// TIA Portal V20 export
FUNCTION_BLOCK "Sequence_1_TopTapeLoading"   // FB32851, LAD
TITLE = Sequence
// Sequence template programmend in ladder logic
// stored: IsIECCheckEnabled true, MemoryReserve 100, Namespace Unit1.Em3, SetENOAutomatically true
   VAR_INPUT
      unitStatus : "LAF_typeUnitStatus";
   END_VAR
   VAR
      instSequenceLADControl { ExternalWritable := 'False'} : "LAF_ControlLadSequence";
      instSequenceLADStatus { ExternalWritable := 'False'} : "LAF_StatusLadSequence";
      statTonTime { ExternalWritable := 'False'} : Array[0..9999] of TON_TIME;
   END_VAR
   VAR_TEMP
      tempCustomerAction : Bool;   // Placeholder for possible actions
      tempDo_nothing_and_wait_for_init : Bool;   // Placeholder for doing nothing
      tempSafeStateCondition : Bool;   // Temp Condition for the equipment module to be in a safe state
   END_VAR
   VAR CONSTANT
      delayTime : Time := T#100ms;
      lowDelayTime : Time := T#1000ms;
      STEP_IDLE : DInt := 1;
      JOB_1_STEP_01 : DInt := 101;
      JOB_1_STEP_10 : DInt := 110;
      JOB_1_STEP_20 : DInt := 120;
      JOB_1_STEP_30 : DInt := 130;
      JOB_1_STEP_40 : DInt := 140;
      JOB_1_STEP_50 : DInt := 150;
      JOB_1_STEP_60 : DInt := 160;
      JOB_1_STEP_70 : DInt := 170;
      JOB_1_STEP_80 : DInt := 180;
      JOB_1_STEP_90 : DInt := 190;
      JOB_2_STEP_01 : DInt := 201;
      JOB_2_STEP_10 : DInt := 210;
      JOB_2_STEP_20 : DInt := 220;
      JOB_2_STEP_30 : DInt := 230;
      JOB_2_STEP_40 : DInt := 240;
      JOB_2_STEP_50 : DInt := 250;
      JOB_2_STEP_60 : DInt := 260;
      JOB_2_STEP_70 : DInt := 270;
      JOB_2_STEP_80 : DInt := 280;
      JOB_2_STEP_90 : DInt := 290;
      JOB_3_STEP_01 : DInt := 301;
      JOB_3_STEP_10 : DInt := 310;
      JOB_3_STEP_20 : DInt := 320;
      JOB_3_STEP_30 : DInt := 330;
      JOB_3_STEP_40 : DInt := 340;
      JOB_3_STEP_50 : DInt := 350;
      JOB_3_STEP_60 : DInt := 360;
      JOB_3_STEP_70 : DInt := 370;
      JOB_3_STEP_80 : DInt := 380;
      JOB_3_STEP_90 : DInt := 390;
      STEP_IMMEDIATE_STOP : DInt := 9001;   // Step executed when an immediate stop command is triggered for the sequence (i.e. when unit is in state aborting)
      TO_DO_INSERT_ACTIONS_HERE : Bool := TRUE;   // Template : Add actions
      TO_DO_INSERT_CONDITION_FOR_TRANSITION_HERE : Bool := TRUE;   // Template : Add conditions
   END_VAR
   VAR_TEMP   // added for the SCL form of the ladder/FBD networks
      _w1 : Bool;
      _w2 : Bool;
   END_VAR
BEGIN

REGION Network 1: BLOCK INFO HEADER
   // (company) / (C) Copyright (year)
   // ---------------------------------------------------------------------------------
   // Title:                             (Title of this block)
   // Comment/Function: (that is implemented in the block)
   // Library/Family:           (that the source is dedicated to)
   // Author:                        (department / person in charge / contact)
   // Target System:          (test system with FW version)
   // Engineering:              TIA Portal (SW version)
   // Restrictions:               (OB types, etc.)
   // Requirements:           (hardware, technological package, etc.)
   // ---------------------------------------------------------------------------------
   // Change log table:
   // Version          | Date             | Signature      | Expert in charge  | Changes applied ------------------------|----------------------|-------------------------|--------------------------------|-----------------------
   // 001.000.000 | yyyy-mm-dd | 0x00000000 | (name of expert) | First released version
END_REGION

REGION Network 2: DESCRIPTION
   // This is a template block provided by the Automation Framework. It can be used to create an own project.
   // The Block Info Header is prepared to put in your own data.
   // Description of the block could be added here and the docu created by Code2Docu.
END_REGION

REGION Network 3: *************** CONTROL **********************
END_REGION

REGION Network 4: Sequence Control ("Enter your Sequins number here")
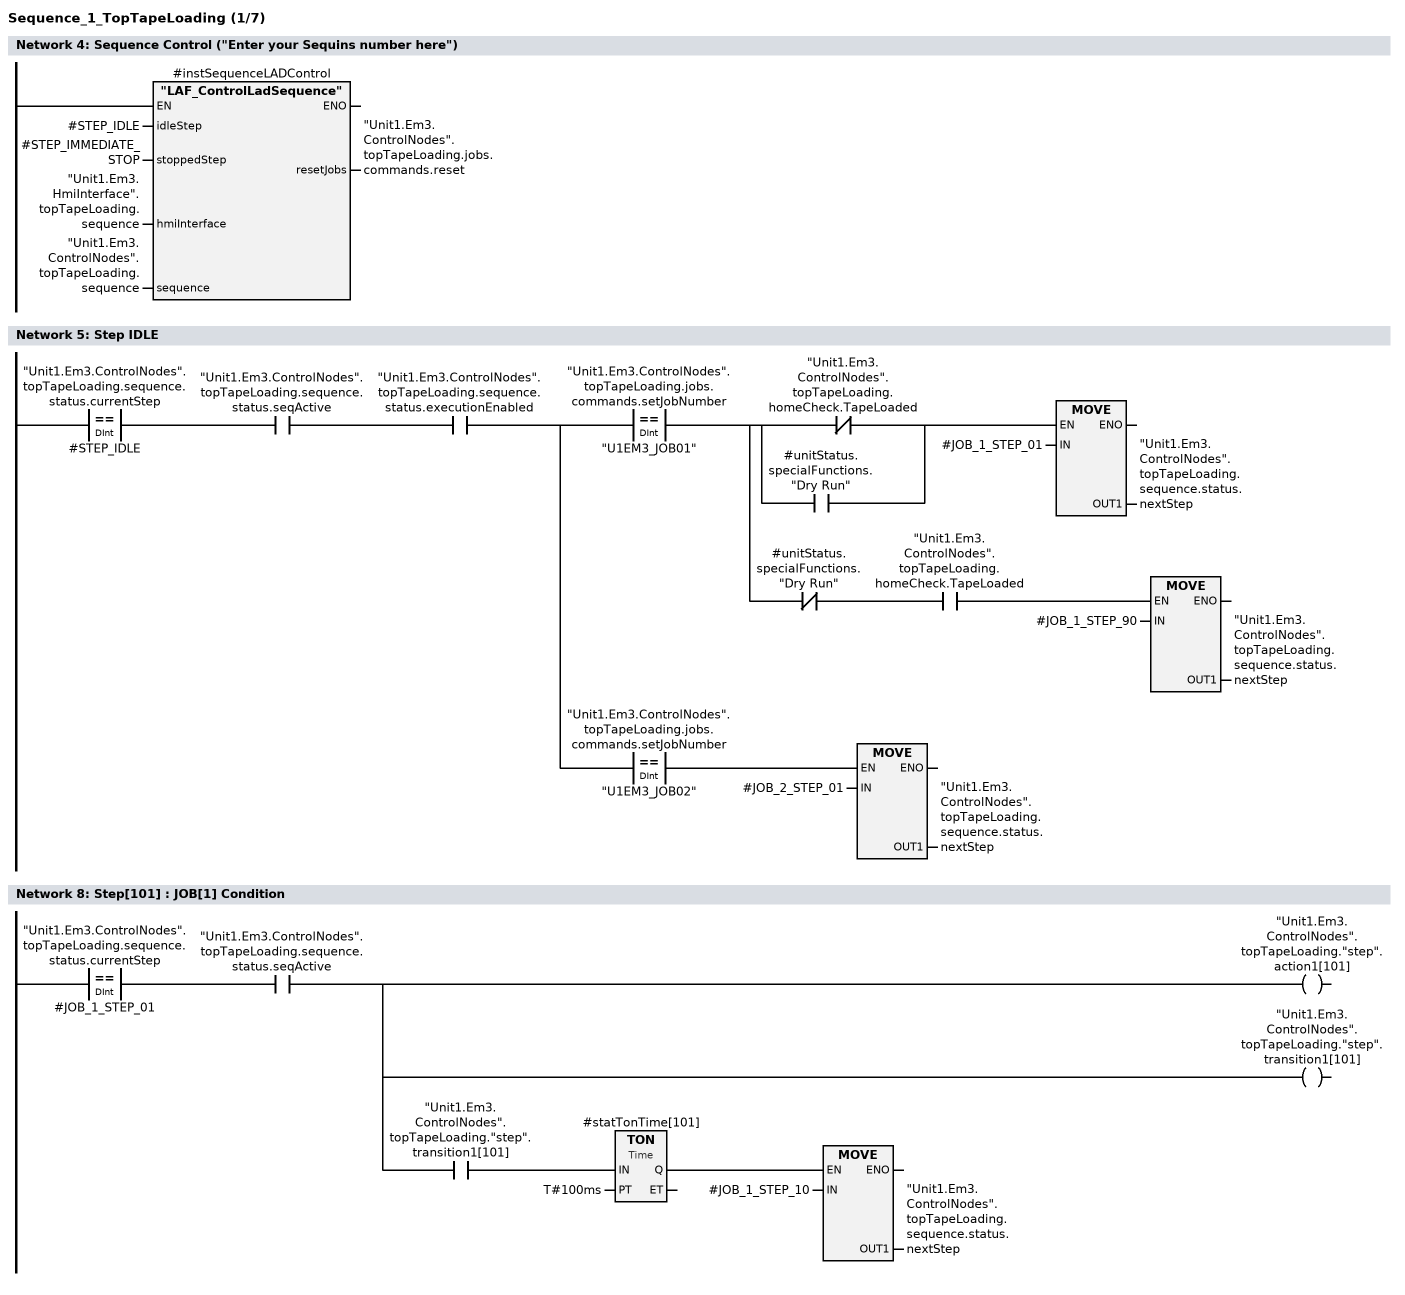
   RUNG wire#powerrail
      #instSequenceLADControl(idleStep := #STEP_IDLE, stoppedStep := #STEP_IMMEDIATE_STOP, hmiInterface := "Unit1.Em3.HmiInterface".topTapeLoading.sequence, sequence := "Unit1.Em3.ControlNodes".topTapeLoading.sequence, resetJobs => "Unit1.Em3.ControlNodes".topTapeLoading.jobs.commands.reset)
   END_RUNG
   // the same network as SCL:
   #instSequenceLADControl(idleStep := #STEP_IDLE,   // "LAF_ControlLadSequence"
                           stoppedStep := #STEP_IMMEDIATE_STOP,
                           hmiInterface := "Unit1.Em3.HmiInterface".topTapeLoading.sequence,
                           sequence := "Unit1.Em3.ControlNodes".topTapeLoading.sequence,
                           resetJobs => "Unit1.Em3.ControlNodes".topTapeLoading.jobs.commands.reset);
END_REGION

REGION Network 5: Step IDLE
   RUNG wire#powerrail
      { S7_Templates := "SrcType := DInt" } EQ_Contact(in1 := "Unit1.Em3.ControlNodes".topTapeLoading.sequence.status.currentStep, in2 := #STEP_IDLE)
      Contact( "Unit1.Em3.ControlNodes".topTapeLoading.sequence.status.seqActive )
      Contact( "Unit1.Em3.ControlNodes".topTapeLoading.sequence.status.executionEnabled )
      wire#w1
      { S7_Templates := "SrcType := DInt" } EQ_Contact(in1 := "Unit1.Em3.ControlNodes".topTapeLoading.jobs.commands.setJobNumber, in2 := "U1EM3_JOB01")
      wire#w2
      I_Contact( "Unit1.Em3.ControlNodes".topTapeLoading.homeCheck.TapeLoaded )
      wire#w3
      Move(in := #JOB_1_STEP_01, out1 => "Unit1.Em3.ControlNodes".topTapeLoading.sequence.status.nextStep)
   END_RUNG
   RUNG wire#w2
      Contact( #unitStatus.specialFunctions."Dry Run" )
   END_RUNG wire#w3
   RUNG wire#w2
      I_Contact( #unitStatus.specialFunctions."Dry Run" )
      Contact( "Unit1.Em3.ControlNodes".topTapeLoading.homeCheck.TapeLoaded )
      Move(in := #JOB_1_STEP_90, out1 => "Unit1.Em3.ControlNodes".topTapeLoading.sequence.status.nextStep)
   END_RUNG
   RUNG wire#w1
      { S7_Templates := "SrcType := DInt" } EQ_Contact(in1 := "Unit1.Em3.ControlNodes".topTapeLoading.jobs.commands.setJobNumber, in2 := "U1EM3_JOB02")
      Move(in := #JOB_2_STEP_01, out1 => "Unit1.Em3.ControlNodes".topTapeLoading.sequence.status.nextStep)
   END_RUNG
   // the same network as SCL:
   #_w1 := ("Unit1.Em3.ControlNodes".topTapeLoading.sequence.status.currentStep = #STEP_IDLE) AND "Unit1.Em3.ControlNodes".topTapeLoading.sequence.status.seqActive AND "Unit1.Em3.ControlNodes".topTapeLoading.sequence.status.executionEnabled;
   #_w2 := #_w1 AND ("Unit1.Em3.ControlNodes".topTapeLoading.jobs.commands.setJobNumber = "U1EM3_JOB01");
   IF #_w2 AND (NOT "Unit1.Em3.ControlNodes".topTapeLoading.homeCheck.TapeLoaded OR #unitStatus.specialFunctions."Dry Run") THEN
       "Unit1.Em3.ControlNodes".topTapeLoading.sequence.status.nextStep := #JOB_1_STEP_01;
   END_IF;
   IF #_w2 AND NOT #unitStatus.specialFunctions."Dry Run" AND "Unit1.Em3.ControlNodes".topTapeLoading.homeCheck.TapeLoaded THEN
       "Unit1.Em3.ControlNodes".topTapeLoading.sequence.status.nextStep := #JOB_1_STEP_90;
   END_IF;
   IF #_w1 AND ("Unit1.Em3.ControlNodes".topTapeLoading.jobs.commands.setJobNumber = "U1EM3_JOB02") THEN
       "Unit1.Em3.ControlNodes".topTapeLoading.sequence.status.nextStep := #JOB_2_STEP_01;
   END_IF;
END_REGION

REGION Network 7: *************** JOB[1] HOMING *************************
END_REGION

REGION Network 8: Step[101] : JOB[1] Condition
   RUNG wire#powerrail
      { S7_Templates := "SrcType := DInt" } EQ_Contact(in1 := "Unit1.Em3.ControlNodes".topTapeLoading.sequence.status.currentStep, in2 := #JOB_1_STEP_01)
      Contact( "Unit1.Em3.ControlNodes".topTapeLoading.sequence.status.seqActive )
      wire#w1
      Coil( "Unit1.Em3.ControlNodes".topTapeLoading."step".action1[101] )
   END_RUNG
   RUNG wire#w1
      Coil( "Unit1.Em3.ControlNodes".topTapeLoading."step".transition1[101] )
   END_RUNG
   RUNG wire#w1
      Contact( "Unit1.Em3.ControlNodes".topTapeLoading."step".transition1[101] )
      { S7_Templates := "time_type := Time" } #statTonTime[101].TON(pt := T#100ms, et =>)
      Move(in := #JOB_1_STEP_10, out1 => "Unit1.Em3.ControlNodes".topTapeLoading.sequence.status.nextStep)
   END_RUNG
   // the same network as SCL:
   "Unit1.Em3.ControlNodes".topTapeLoading."step".action1[101] := ("Unit1.Em3.ControlNodes".topTapeLoading.sequence.status.currentStep = #JOB_1_STEP_01) AND "Unit1.Em3.ControlNodes".topTapeLoading.sequence.status.seqActive;
   "Unit1.Em3.ControlNodes".topTapeLoading."step".transition1[101] := ("Unit1.Em3.ControlNodes".topTapeLoading.sequence.status.currentStep = #JOB_1_STEP_01) AND "Unit1.Em3.ControlNodes".topTapeLoading.sequence.status.seqActive;
   #statTonTime[101].TON(IN := ("Unit1.Em3.ControlNodes".topTapeLoading.sequence.status.currentStep = #JOB_1_STEP_01) AND "Unit1.Em3.ControlNodes".topTapeLoading.sequence.status.seqActive AND "Unit1.Em3.ControlNodes".topTapeLoading."step".transition1[101],
                         PT := T#100ms);
   IF #statTonTime[101].Q THEN
       "Unit1.Em3.ControlNodes".topTapeLoading.sequence.status.nextStep := #JOB_1_STEP_10;
   END_IF;
END_REGION

REGION Network 9: Step[110] : Top Tape Loading Backward
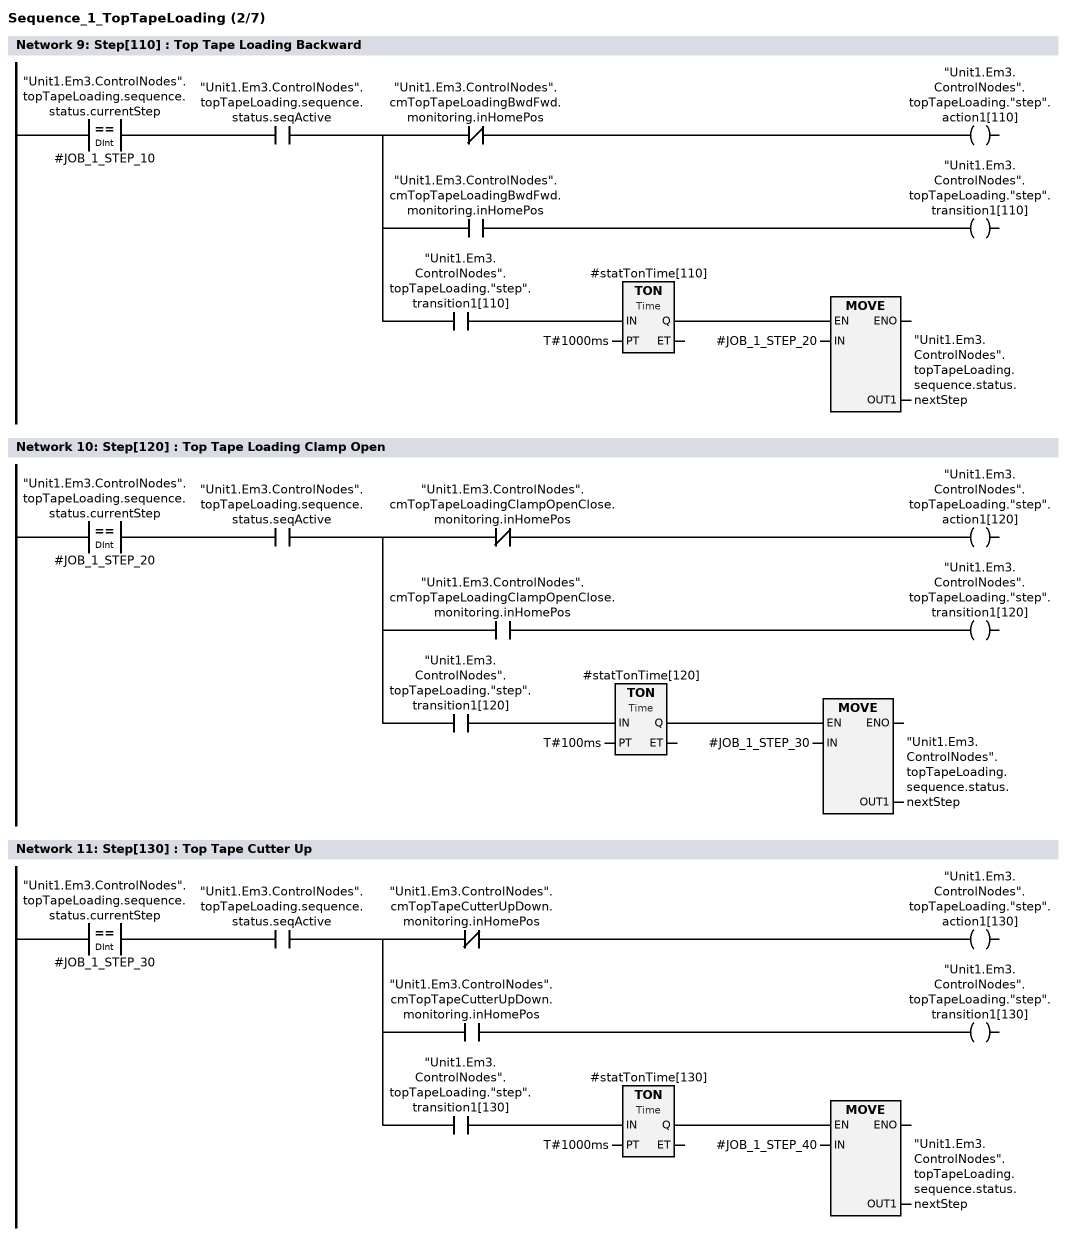
   RUNG wire#powerrail
      { S7_Templates := "SrcType := DInt" } EQ_Contact(in1 := "Unit1.Em3.ControlNodes".topTapeLoading.sequence.status.currentStep, in2 := #JOB_1_STEP_10)
      Contact( "Unit1.Em3.ControlNodes".topTapeLoading.sequence.status.seqActive )
      wire#w1
      I_Contact( "Unit1.Em3.ControlNodes".cmTopTapeLoadingBwdFwd.monitoring.inHomePos )
      Coil( "Unit1.Em3.ControlNodes".topTapeLoading."step".action1[110] )
   END_RUNG
   RUNG wire#w1
      Contact( "Unit1.Em3.ControlNodes".cmTopTapeLoadingBwdFwd.monitoring.inHomePos )
      Coil( "Unit1.Em3.ControlNodes".topTapeLoading."step".transition1[110] )
   END_RUNG
   RUNG wire#w1
      Contact( "Unit1.Em3.ControlNodes".topTapeLoading."step".transition1[110] )
      { S7_Templates := "time_type := Time" } #statTonTime[110].TON(pt := T#1000ms, et =>)
      Move(in := #JOB_1_STEP_20, out1 => "Unit1.Em3.ControlNodes".topTapeLoading.sequence.status.nextStep)
   END_RUNG
   // the same network as SCL:
   #_w1 := ("Unit1.Em3.ControlNodes".topTapeLoading.sequence.status.currentStep = #JOB_1_STEP_10) AND "Unit1.Em3.ControlNodes".topTapeLoading.sequence.status.seqActive;
   "Unit1.Em3.ControlNodes".topTapeLoading."step".action1[110] := #_w1 AND NOT "Unit1.Em3.ControlNodes".cmTopTapeLoadingBwdFwd.monitoring.inHomePos;
   "Unit1.Em3.ControlNodes".topTapeLoading."step".transition1[110] := #_w1 AND "Unit1.Em3.ControlNodes".cmTopTapeLoadingBwdFwd.monitoring.inHomePos;
   #statTonTime[110].TON(IN := #_w1 AND "Unit1.Em3.ControlNodes".topTapeLoading."step".transition1[110],
                         PT := T#1000ms);
   IF #statTonTime[110].Q THEN
       "Unit1.Em3.ControlNodes".topTapeLoading.sequence.status.nextStep := #JOB_1_STEP_20;
   END_IF;
END_REGION

REGION Network 10: Step[120] : Top Tape Loading Clamp Open
   RUNG wire#powerrail
      { S7_Templates := "SrcType := DInt" } EQ_Contact(in1 := "Unit1.Em3.ControlNodes".topTapeLoading.sequence.status.currentStep, in2 := #JOB_1_STEP_20)
      Contact( "Unit1.Em3.ControlNodes".topTapeLoading.sequence.status.seqActive )
      wire#w1
      I_Contact( "Unit1.Em3.ControlNodes".cmTopTapeLoadingClampOpenClose.monitoring.inHomePos )
      Coil( "Unit1.Em3.ControlNodes".topTapeLoading."step".action1[120] )
   END_RUNG
   RUNG wire#w1
      Contact( "Unit1.Em3.ControlNodes".cmTopTapeLoadingClampOpenClose.monitoring.inHomePos )
      Coil( "Unit1.Em3.ControlNodes".topTapeLoading."step".transition1[120] )
   END_RUNG
   RUNG wire#w1
      Contact( "Unit1.Em3.ControlNodes".topTapeLoading."step".transition1[120] )
      { S7_Templates := "time_type := Time" } #statTonTime[120].TON(pt := T#100ms, et =>)
      Move(in := #JOB_1_STEP_30, out1 => "Unit1.Em3.ControlNodes".topTapeLoading.sequence.status.nextStep)
   END_RUNG
   // the same network as SCL:
   #_w1 := ("Unit1.Em3.ControlNodes".topTapeLoading.sequence.status.currentStep = #JOB_1_STEP_20) AND "Unit1.Em3.ControlNodes".topTapeLoading.sequence.status.seqActive;
   "Unit1.Em3.ControlNodes".topTapeLoading."step".action1[120] := #_w1 AND NOT "Unit1.Em3.ControlNodes".cmTopTapeLoadingClampOpenClose.monitoring.inHomePos;
   "Unit1.Em3.ControlNodes".topTapeLoading."step".transition1[120] := #_w1 AND "Unit1.Em3.ControlNodes".cmTopTapeLoadingClampOpenClose.monitoring.inHomePos;
   #statTonTime[120].TON(IN := #_w1 AND "Unit1.Em3.ControlNodes".topTapeLoading."step".transition1[120],
                         PT := T#100ms);
   IF #statTonTime[120].Q THEN
       "Unit1.Em3.ControlNodes".topTapeLoading.sequence.status.nextStep := #JOB_1_STEP_30;
   END_IF;
END_REGION

REGION Network 11: Step[130] : Top Tape Cutter Up
   RUNG wire#powerrail
      { S7_Templates := "SrcType := DInt" } EQ_Contact(in1 := "Unit1.Em3.ControlNodes".topTapeLoading.sequence.status.currentStep, in2 := #JOB_1_STEP_30)
      Contact( "Unit1.Em3.ControlNodes".topTapeLoading.sequence.status.seqActive )
      wire#w1
      I_Contact( "Unit1.Em3.ControlNodes".cmTopTapeCutterUpDown.monitoring.inHomePos )
      Coil( "Unit1.Em3.ControlNodes".topTapeLoading."step".action1[130] )
   END_RUNG
   RUNG wire#w1
      Contact( "Unit1.Em3.ControlNodes".cmTopTapeCutterUpDown.monitoring.inHomePos )
      Coil( "Unit1.Em3.ControlNodes".topTapeLoading."step".transition1[130] )
   END_RUNG
   RUNG wire#w1
      Contact( "Unit1.Em3.ControlNodes".topTapeLoading."step".transition1[130] )
      { S7_Templates := "time_type := Time" } #statTonTime[130].TON(pt := T#1000ms, et =>)
      Move(in := #JOB_1_STEP_40, out1 => "Unit1.Em3.ControlNodes".topTapeLoading.sequence.status.nextStep)
   END_RUNG
   // the same network as SCL:
   #_w1 := ("Unit1.Em3.ControlNodes".topTapeLoading.sequence.status.currentStep = #JOB_1_STEP_30) AND "Unit1.Em3.ControlNodes".topTapeLoading.sequence.status.seqActive;
   "Unit1.Em3.ControlNodes".topTapeLoading."step".action1[130] := #_w1 AND NOT "Unit1.Em3.ControlNodes".cmTopTapeCutterUpDown.monitoring.inHomePos;
   "Unit1.Em3.ControlNodes".topTapeLoading."step".transition1[130] := #_w1 AND "Unit1.Em3.ControlNodes".cmTopTapeCutterUpDown.monitoring.inHomePos;
   #statTonTime[130].TON(IN := #_w1 AND "Unit1.Em3.ControlNodes".topTapeLoading."step".transition1[130],
                         PT := T#1000ms);
   IF #statTonTime[130].Q THEN
       "Unit1.Em3.ControlNodes".topTapeLoading.sequence.status.nextStep := #JOB_1_STEP_40;
   END_IF;
END_REGION

REGION Network 12: Step[140] : Top Tape Cutter Clamp Down
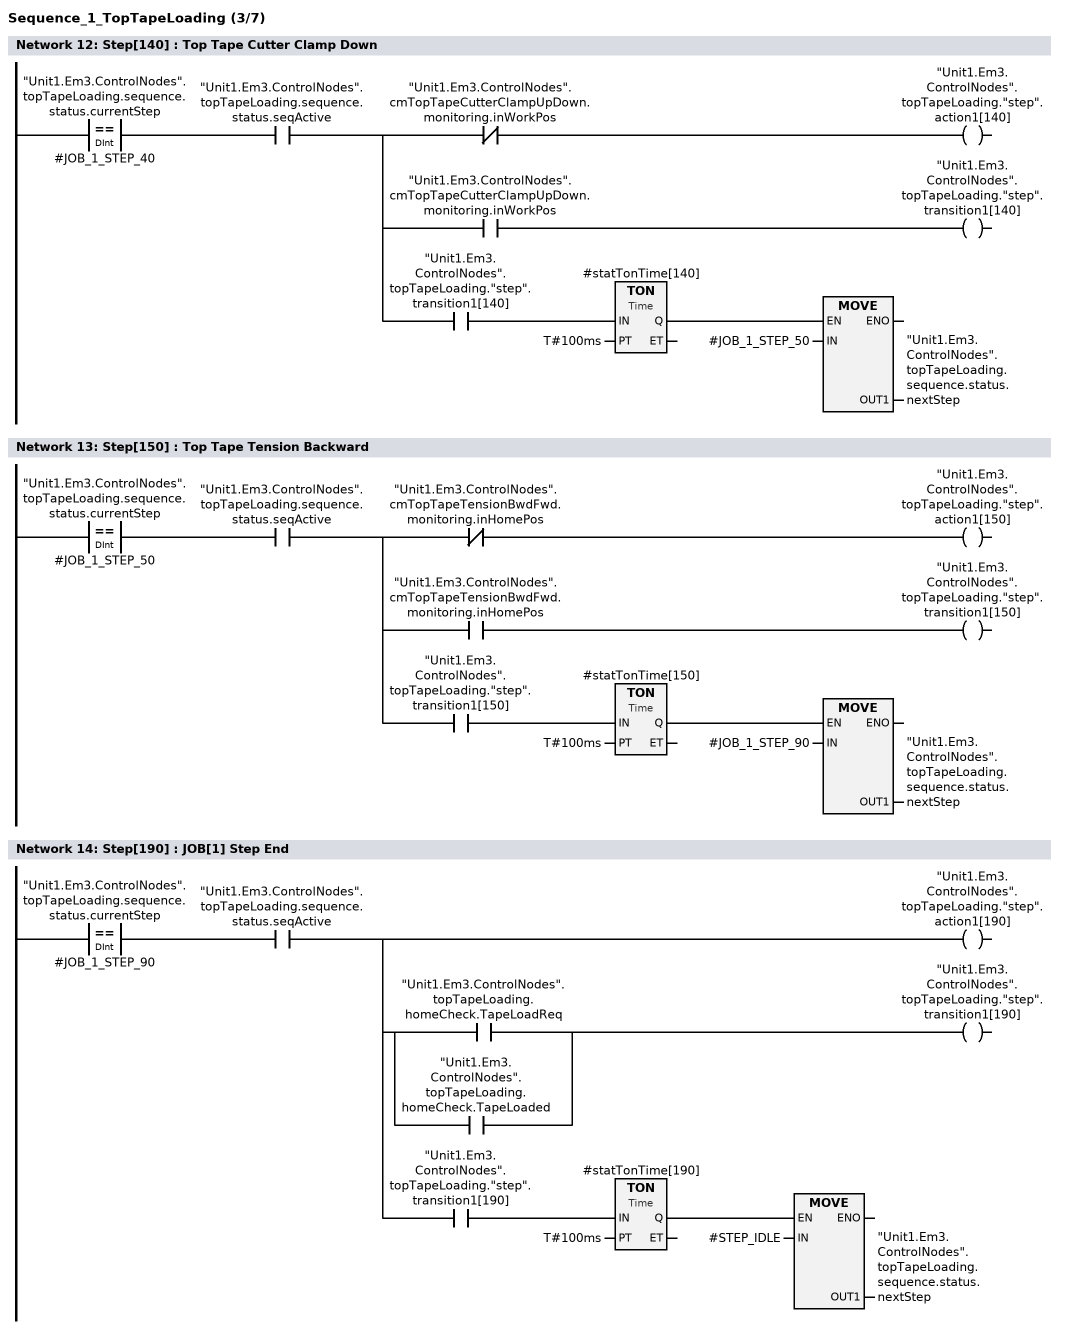
   RUNG wire#powerrail
      { S7_Templates := "SrcType := DInt" } EQ_Contact(in1 := "Unit1.Em3.ControlNodes".topTapeLoading.sequence.status.currentStep, in2 := #JOB_1_STEP_40)
      Contact( "Unit1.Em3.ControlNodes".topTapeLoading.sequence.status.seqActive )
      wire#w1
      I_Contact( "Unit1.Em3.ControlNodes".cmTopTapeCutterClampUpDown.monitoring.inWorkPos )
      Coil( "Unit1.Em3.ControlNodes".topTapeLoading."step".action1[140] )
   END_RUNG
   RUNG wire#w1
      Contact( "Unit1.Em3.ControlNodes".cmTopTapeCutterClampUpDown.monitoring.inWorkPos )
      Coil( "Unit1.Em3.ControlNodes".topTapeLoading."step".transition1[140] )
   END_RUNG
   RUNG wire#w1
      Contact( "Unit1.Em3.ControlNodes".topTapeLoading."step".transition1[140] )
      { S7_Templates := "time_type := Time" } #statTonTime[140].TON(pt := T#100ms, et =>)
      Move(in := #JOB_1_STEP_50, out1 => "Unit1.Em3.ControlNodes".topTapeLoading.sequence.status.nextStep)
   END_RUNG
   // the same network as SCL:
   #_w1 := ("Unit1.Em3.ControlNodes".topTapeLoading.sequence.status.currentStep = #JOB_1_STEP_40) AND "Unit1.Em3.ControlNodes".topTapeLoading.sequence.status.seqActive;
   "Unit1.Em3.ControlNodes".topTapeLoading."step".action1[140] := #_w1 AND NOT "Unit1.Em3.ControlNodes".cmTopTapeCutterClampUpDown.monitoring.inWorkPos;
   "Unit1.Em3.ControlNodes".topTapeLoading."step".transition1[140] := #_w1 AND "Unit1.Em3.ControlNodes".cmTopTapeCutterClampUpDown.monitoring.inWorkPos;
   #statTonTime[140].TON(IN := #_w1 AND "Unit1.Em3.ControlNodes".topTapeLoading."step".transition1[140],
                         PT := T#100ms);
   IF #statTonTime[140].Q THEN
       "Unit1.Em3.ControlNodes".topTapeLoading.sequence.status.nextStep := #JOB_1_STEP_50;
   END_IF;
END_REGION

REGION Network 13: Step[150] : Top Tape Tension Backward
   RUNG wire#powerrail
      { S7_Templates := "SrcType := DInt" } EQ_Contact(in1 := "Unit1.Em3.ControlNodes".topTapeLoading.sequence.status.currentStep, in2 := #JOB_1_STEP_50)
      Contact( "Unit1.Em3.ControlNodes".topTapeLoading.sequence.status.seqActive )
      wire#w1
      I_Contact( "Unit1.Em3.ControlNodes".cmTopTapeTensionBwdFwd.monitoring.inHomePos )
      Coil( "Unit1.Em3.ControlNodes".topTapeLoading."step".action1[150] )
   END_RUNG
   RUNG wire#w1
      Contact( "Unit1.Em3.ControlNodes".cmTopTapeTensionBwdFwd.monitoring.inHomePos )
      Coil( "Unit1.Em3.ControlNodes".topTapeLoading."step".transition1[150] )
   END_RUNG
   RUNG wire#w1
      Contact( "Unit1.Em3.ControlNodes".topTapeLoading."step".transition1[150] )
      { S7_Templates := "time_type := Time" } #statTonTime[150].TON(pt := T#100ms, et =>)
      Move(in := #JOB_1_STEP_90, out1 => "Unit1.Em3.ControlNodes".topTapeLoading.sequence.status.nextStep)
   END_RUNG
   // the same network as SCL:
   #_w1 := ("Unit1.Em3.ControlNodes".topTapeLoading.sequence.status.currentStep = #JOB_1_STEP_50) AND "Unit1.Em3.ControlNodes".topTapeLoading.sequence.status.seqActive;
   "Unit1.Em3.ControlNodes".topTapeLoading."step".action1[150] := #_w1 AND NOT "Unit1.Em3.ControlNodes".cmTopTapeTensionBwdFwd.monitoring.inHomePos;
   "Unit1.Em3.ControlNodes".topTapeLoading."step".transition1[150] := #_w1 AND "Unit1.Em3.ControlNodes".cmTopTapeTensionBwdFwd.monitoring.inHomePos;
   #statTonTime[150].TON(IN := #_w1 AND "Unit1.Em3.ControlNodes".topTapeLoading."step".transition1[150],
                         PT := T#100ms);
   IF #statTonTime[150].Q THEN
       "Unit1.Em3.ControlNodes".topTapeLoading.sequence.status.nextStep := #JOB_1_STEP_90;
   END_IF;
END_REGION

REGION Network 14: Step[190] : JOB[1] Step End
   RUNG wire#powerrail
      { S7_Templates := "SrcType := DInt" } EQ_Contact(in1 := "Unit1.Em3.ControlNodes".topTapeLoading.sequence.status.currentStep, in2 := #JOB_1_STEP_90)
      Contact( "Unit1.Em3.ControlNodes".topTapeLoading.sequence.status.seqActive )
      wire#w1
      Coil( "Unit1.Em3.ControlNodes".topTapeLoading."step".action1[190] )
   END_RUNG
   RUNG wire#w1
      Contact( "Unit1.Em3.ControlNodes".topTapeLoading.homeCheck.TapeLoadReq )
      wire#w2
      Coil( "Unit1.Em3.ControlNodes".topTapeLoading."step".transition1[190] )
   END_RUNG
   RUNG wire#w1
      Contact( "Unit1.Em3.ControlNodes".topTapeLoading.homeCheck.TapeLoaded )
   END_RUNG wire#w2
   RUNG wire#w1
      Contact( "Unit1.Em3.ControlNodes".topTapeLoading."step".transition1[190] )
      { S7_Templates := "time_type := Time" } #statTonTime[190].TON(pt := T#100ms, et =>)
      Move(in := #STEP_IDLE, out1 => "Unit1.Em3.ControlNodes".topTapeLoading.sequence.status.nextStep)
   END_RUNG
   // the same network as SCL:
   "Unit1.Em3.ControlNodes".topTapeLoading."step".action1[190] := ("Unit1.Em3.ControlNodes".topTapeLoading.sequence.status.currentStep = #JOB_1_STEP_90) AND "Unit1.Em3.ControlNodes".topTapeLoading.sequence.status.seqActive;
   "Unit1.Em3.ControlNodes".topTapeLoading."step".transition1[190] := ("Unit1.Em3.ControlNodes".topTapeLoading.sequence.status.currentStep = #JOB_1_STEP_90) AND "Unit1.Em3.ControlNodes".topTapeLoading.sequence.status.seqActive AND ("Unit1.Em3.ControlNodes".topTapeLoading.homeCheck.TapeLoadReq OR "Unit1.Em3.ControlNodes".topTapeLoading.homeCheck.TapeLoaded);
   #statTonTime[190].TON(IN := ("Unit1.Em3.ControlNodes".topTapeLoading.sequence.status.currentStep = #JOB_1_STEP_90) AND "Unit1.Em3.ControlNodes".topTapeLoading.sequence.status.seqActive AND "Unit1.Em3.ControlNodes".topTapeLoading."step".transition1[190],
                         PT := T#100ms);
   IF #statTonTime[190].Q THEN
       "Unit1.Em3.ControlNodes".topTapeLoading.sequence.status.nextStep := #STEP_IDLE;
   END_IF;
END_REGION

REGION Network 15: *************** JOB[2] TOP TAPE CHARGE=AUTO *************************
END_REGION

REGION Network 16: Step[201] : JOB[2] Condition
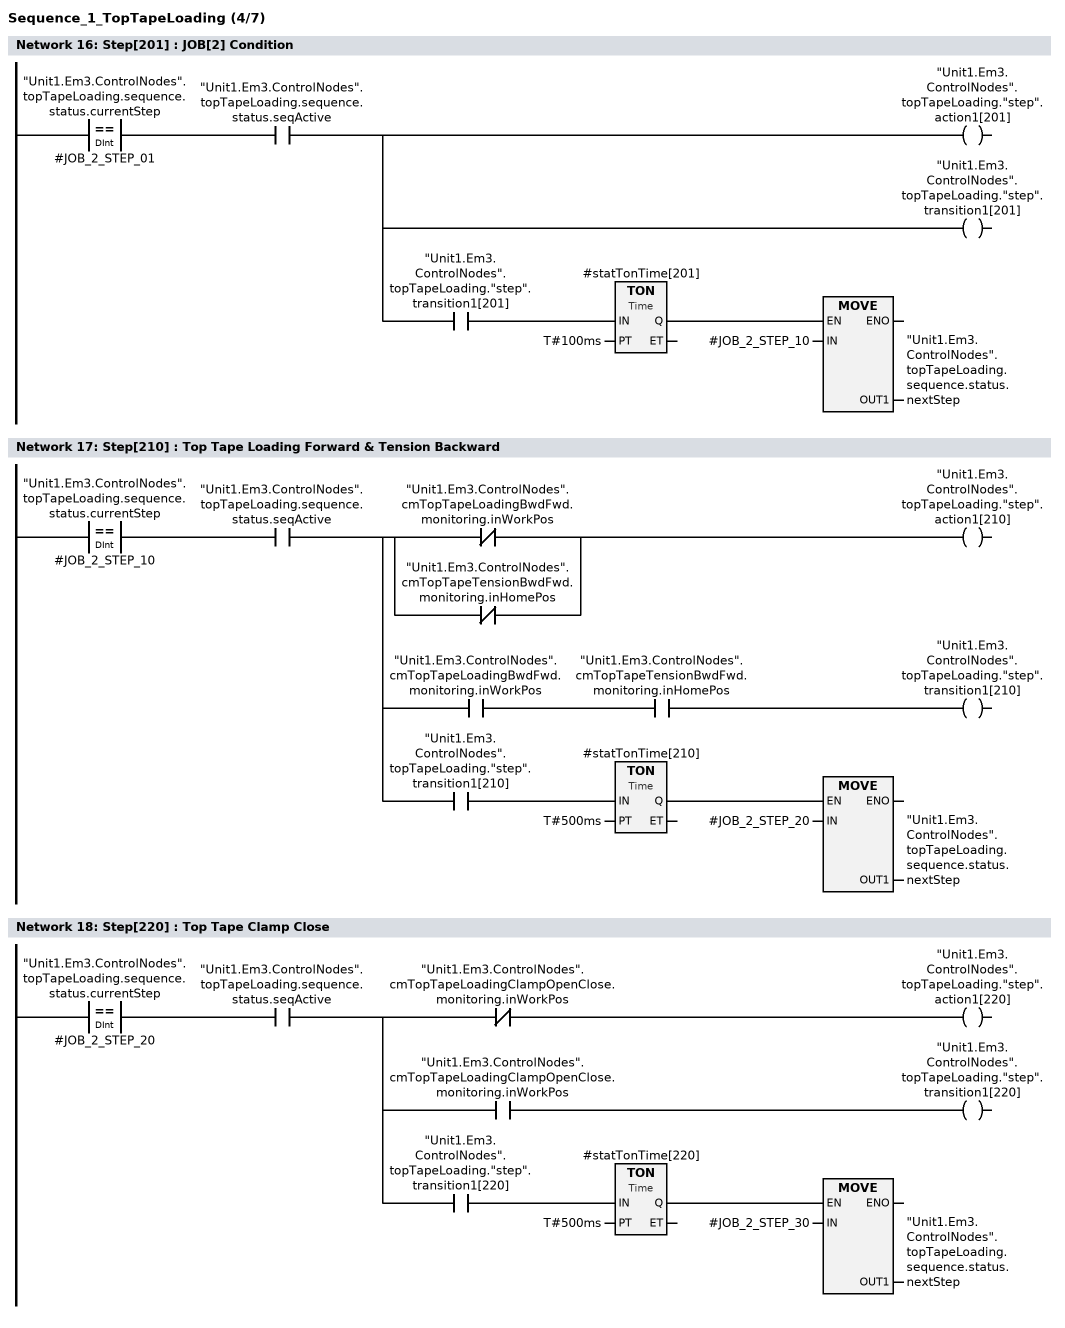
   RUNG wire#powerrail
      { S7_Templates := "SrcType := DInt" } EQ_Contact(in1 := "Unit1.Em3.ControlNodes".topTapeLoading.sequence.status.currentStep, in2 := #JOB_2_STEP_01)
      Contact( "Unit1.Em3.ControlNodes".topTapeLoading.sequence.status.seqActive )
      wire#w1
      Coil( "Unit1.Em3.ControlNodes".topTapeLoading."step".action1[201] )
   END_RUNG
   RUNG wire#w1
      Coil( "Unit1.Em3.ControlNodes".topTapeLoading."step".transition1[201] )
   END_RUNG
   RUNG wire#w1
      Contact( "Unit1.Em3.ControlNodes".topTapeLoading."step".transition1[201] )
      { S7_Templates := "time_type := Time" } #statTonTime[201].TON(pt := T#100ms, et =>)
      Move(in := #JOB_2_STEP_10, out1 => "Unit1.Em3.ControlNodes".topTapeLoading.sequence.status.nextStep)
   END_RUNG
   // the same network as SCL:
   "Unit1.Em3.ControlNodes".topTapeLoading."step".action1[201] := ("Unit1.Em3.ControlNodes".topTapeLoading.sequence.status.currentStep = #JOB_2_STEP_01) AND "Unit1.Em3.ControlNodes".topTapeLoading.sequence.status.seqActive;
   "Unit1.Em3.ControlNodes".topTapeLoading."step".transition1[201] := ("Unit1.Em3.ControlNodes".topTapeLoading.sequence.status.currentStep = #JOB_2_STEP_01) AND "Unit1.Em3.ControlNodes".topTapeLoading.sequence.status.seqActive;
   #statTonTime[201].TON(IN := ("Unit1.Em3.ControlNodes".topTapeLoading.sequence.status.currentStep = #JOB_2_STEP_01) AND "Unit1.Em3.ControlNodes".topTapeLoading.sequence.status.seqActive AND "Unit1.Em3.ControlNodes".topTapeLoading."step".transition1[201],
                         PT := T#100ms);
   IF #statTonTime[201].Q THEN
       "Unit1.Em3.ControlNodes".topTapeLoading.sequence.status.nextStep := #JOB_2_STEP_10;
   END_IF;
END_REGION

REGION Network 17: Step[210] : Top Tape Loading Forward & Tension Backward
   RUNG wire#powerrail
      { S7_Templates := "SrcType := DInt" } EQ_Contact(in1 := "Unit1.Em3.ControlNodes".topTapeLoading.sequence.status.currentStep, in2 := #JOB_2_STEP_10)
      Contact( "Unit1.Em3.ControlNodes".topTapeLoading.sequence.status.seqActive )
      wire#w1
      I_Contact( "Unit1.Em3.ControlNodes".cmTopTapeLoadingBwdFwd.monitoring.inWorkPos )
      wire#w2
      Coil( "Unit1.Em3.ControlNodes".topTapeLoading."step".action1[210] )
   END_RUNG
   RUNG wire#w1
      I_Contact( "Unit1.Em3.ControlNodes".cmTopTapeTensionBwdFwd.monitoring.inHomePos )
   END_RUNG wire#w2
   RUNG wire#w1
      Contact( "Unit1.Em3.ControlNodes".cmTopTapeLoadingBwdFwd.monitoring.inWorkPos )
      Contact( "Unit1.Em3.ControlNodes".cmTopTapeTensionBwdFwd.monitoring.inHomePos )
      Coil( "Unit1.Em3.ControlNodes".topTapeLoading."step".transition1[210] )
   END_RUNG
   RUNG wire#w1
      Contact( "Unit1.Em3.ControlNodes".topTapeLoading."step".transition1[210] )
      { S7_Templates := "time_type := Time" } #statTonTime[210].TON(pt := T#500ms, et =>)
      Move(in := #JOB_2_STEP_20, out1 => "Unit1.Em3.ControlNodes".topTapeLoading.sequence.status.nextStep)
   END_RUNG
   // the same network as SCL:
   #_w1 := ("Unit1.Em3.ControlNodes".topTapeLoading.sequence.status.currentStep = #JOB_2_STEP_10) AND "Unit1.Em3.ControlNodes".topTapeLoading.sequence.status.seqActive;
   "Unit1.Em3.ControlNodes".topTapeLoading."step".action1[210] := #_w1 AND (NOT "Unit1.Em3.ControlNodes".cmTopTapeLoadingBwdFwd.monitoring.inWorkPos OR NOT "Unit1.Em3.ControlNodes".cmTopTapeTensionBwdFwd.monitoring.inHomePos);
   "Unit1.Em3.ControlNodes".topTapeLoading."step".transition1[210] := #_w1 AND "Unit1.Em3.ControlNodes".cmTopTapeLoadingBwdFwd.monitoring.inWorkPos AND "Unit1.Em3.ControlNodes".cmTopTapeTensionBwdFwd.monitoring.inHomePos;
   #statTonTime[210].TON(IN := #_w1 AND "Unit1.Em3.ControlNodes".topTapeLoading."step".transition1[210],
                         PT := T#500ms);
   IF #statTonTime[210].Q THEN
       "Unit1.Em3.ControlNodes".topTapeLoading.sequence.status.nextStep := #JOB_2_STEP_20;
   END_IF;
END_REGION

REGION Network 18: Step[220] : Top Tape Clamp Close
   RUNG wire#powerrail
      { S7_Templates := "SrcType := DInt" } EQ_Contact(in1 := "Unit1.Em3.ControlNodes".topTapeLoading.sequence.status.currentStep, in2 := #JOB_2_STEP_20)
      Contact( "Unit1.Em3.ControlNodes".topTapeLoading.sequence.status.seqActive )
      wire#w1
      I_Contact( "Unit1.Em3.ControlNodes".cmTopTapeLoadingClampOpenClose.monitoring.inWorkPos )
      Coil( "Unit1.Em3.ControlNodes".topTapeLoading."step".action1[220] )
   END_RUNG
   RUNG wire#w1
      Contact( "Unit1.Em3.ControlNodes".cmTopTapeLoadingClampOpenClose.monitoring.inWorkPos )
      Coil( "Unit1.Em3.ControlNodes".topTapeLoading."step".transition1[220] )
   END_RUNG
   RUNG wire#w1
      Contact( "Unit1.Em3.ControlNodes".topTapeLoading."step".transition1[220] )
      { S7_Templates := "time_type := Time" } #statTonTime[220].TON(pt := T#500ms, et =>)
      Move(in := #JOB_2_STEP_30, out1 => "Unit1.Em3.ControlNodes".topTapeLoading.sequence.status.nextStep)
   END_RUNG
   // the same network as SCL:
   #_w1 := ("Unit1.Em3.ControlNodes".topTapeLoading.sequence.status.currentStep = #JOB_2_STEP_20) AND "Unit1.Em3.ControlNodes".topTapeLoading.sequence.status.seqActive;
   "Unit1.Em3.ControlNodes".topTapeLoading."step".action1[220] := #_w1 AND NOT "Unit1.Em3.ControlNodes".cmTopTapeLoadingClampOpenClose.monitoring.inWorkPos;
   "Unit1.Em3.ControlNodes".topTapeLoading."step".transition1[220] := #_w1 AND "Unit1.Em3.ControlNodes".cmTopTapeLoadingClampOpenClose.monitoring.inWorkPos;
   #statTonTime[220].TON(IN := #_w1 AND "Unit1.Em3.ControlNodes".topTapeLoading."step".transition1[220],
                         PT := T#500ms);
   IF #statTonTime[220].Q THEN
       "Unit1.Em3.ControlNodes".topTapeLoading.sequence.status.nextStep := #JOB_2_STEP_30;
   END_IF;
END_REGION

REGION Network 19: Step[230] : Top Tape Cutter Clamp Up
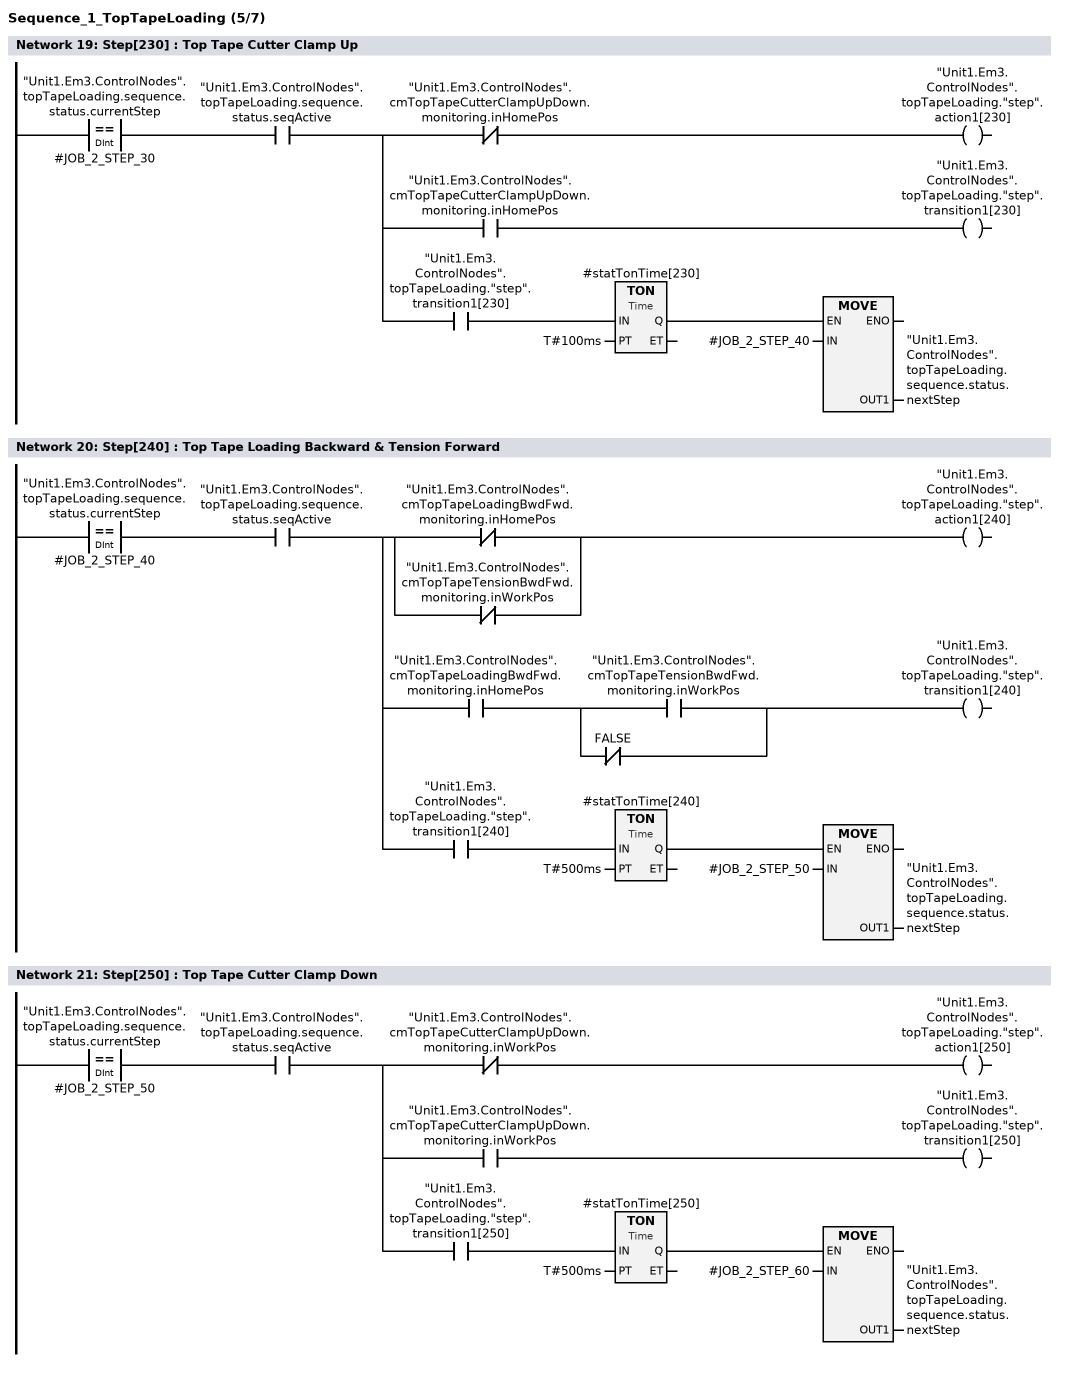
   RUNG wire#powerrail
      { S7_Templates := "SrcType := DInt" } EQ_Contact(in1 := "Unit1.Em3.ControlNodes".topTapeLoading.sequence.status.currentStep, in2 := #JOB_2_STEP_30)
      Contact( "Unit1.Em3.ControlNodes".topTapeLoading.sequence.status.seqActive )
      wire#w1
      I_Contact( "Unit1.Em3.ControlNodes".cmTopTapeCutterClampUpDown.monitoring.inHomePos )
      Coil( "Unit1.Em3.ControlNodes".topTapeLoading."step".action1[230] )
   END_RUNG
   RUNG wire#w1
      Contact( "Unit1.Em3.ControlNodes".cmTopTapeCutterClampUpDown.monitoring.inHomePos )
      Coil( "Unit1.Em3.ControlNodes".topTapeLoading."step".transition1[230] )
   END_RUNG
   RUNG wire#w1
      Contact( "Unit1.Em3.ControlNodes".topTapeLoading."step".transition1[230] )
      { S7_Templates := "time_type := Time" } #statTonTime[230].TON(pt := T#100ms, et =>)
      Move(in := #JOB_2_STEP_40, out1 => "Unit1.Em3.ControlNodes".topTapeLoading.sequence.status.nextStep)
   END_RUNG
   // the same network as SCL:
   #_w1 := ("Unit1.Em3.ControlNodes".topTapeLoading.sequence.status.currentStep = #JOB_2_STEP_30) AND "Unit1.Em3.ControlNodes".topTapeLoading.sequence.status.seqActive;
   "Unit1.Em3.ControlNodes".topTapeLoading."step".action1[230] := #_w1 AND NOT "Unit1.Em3.ControlNodes".cmTopTapeCutterClampUpDown.monitoring.inHomePos;
   "Unit1.Em3.ControlNodes".topTapeLoading."step".transition1[230] := #_w1 AND "Unit1.Em3.ControlNodes".cmTopTapeCutterClampUpDown.monitoring.inHomePos;
   #statTonTime[230].TON(IN := #_w1 AND "Unit1.Em3.ControlNodes".topTapeLoading."step".transition1[230],
                         PT := T#100ms);
   IF #statTonTime[230].Q THEN
       "Unit1.Em3.ControlNodes".topTapeLoading.sequence.status.nextStep := #JOB_2_STEP_40;
   END_IF;
END_REGION

REGION Network 20: Step[240] : Top Tape Loading Backward & Tension Forward
   RUNG wire#powerrail
      { S7_Templates := "SrcType := DInt" } EQ_Contact(in1 := "Unit1.Em3.ControlNodes".topTapeLoading.sequence.status.currentStep, in2 := #JOB_2_STEP_40)
      Contact( "Unit1.Em3.ControlNodes".topTapeLoading.sequence.status.seqActive )
      wire#w1
      I_Contact( "Unit1.Em3.ControlNodes".cmTopTapeLoadingBwdFwd.monitoring.inHomePos )
      wire#w2
      Coil( "Unit1.Em3.ControlNodes".topTapeLoading."step".action1[240] )
   END_RUNG
   RUNG wire#w1
      I_Contact( "Unit1.Em3.ControlNodes".cmTopTapeTensionBwdFwd.monitoring.inWorkPos )
   END_RUNG wire#w2
   RUNG wire#w1
      Contact( "Unit1.Em3.ControlNodes".cmTopTapeLoadingBwdFwd.monitoring.inHomePos )
      wire#w3
      Contact( "Unit1.Em3.ControlNodes".cmTopTapeTensionBwdFwd.monitoring.inWorkPos )
      wire#w4
      Coil( "Unit1.Em3.ControlNodes".topTapeLoading."step".transition1[240] )
   END_RUNG
   RUNG wire#w3
      I_Contact( FALSE )
   END_RUNG wire#w4
   RUNG wire#w1
      Contact( "Unit1.Em3.ControlNodes".topTapeLoading."step".transition1[240] )
      { S7_Templates := "time_type := Time" } #statTonTime[240].TON(pt := T#500ms, et =>)
      Move(in := #JOB_2_STEP_50, out1 => "Unit1.Em3.ControlNodes".topTapeLoading.sequence.status.nextStep)
   END_RUNG
   // the same network as SCL:
   #_w1 := ("Unit1.Em3.ControlNodes".topTapeLoading.sequence.status.currentStep = #JOB_2_STEP_40) AND "Unit1.Em3.ControlNodes".topTapeLoading.sequence.status.seqActive;
   "Unit1.Em3.ControlNodes".topTapeLoading."step".action1[240] := #_w1 AND (NOT "Unit1.Em3.ControlNodes".cmTopTapeLoadingBwdFwd.monitoring.inHomePos OR NOT "Unit1.Em3.ControlNodes".cmTopTapeTensionBwdFwd.monitoring.inWorkPos);
   "Unit1.Em3.ControlNodes".topTapeLoading."step".transition1[240] := #_w1 AND "Unit1.Em3.ControlNodes".cmTopTapeLoadingBwdFwd.monitoring.inHomePos AND ("Unit1.Em3.ControlNodes".cmTopTapeTensionBwdFwd.monitoring.inWorkPos OR NOT FALSE);
   #statTonTime[240].TON(IN := #_w1 AND "Unit1.Em3.ControlNodes".topTapeLoading."step".transition1[240],
                         PT := T#500ms);
   IF #statTonTime[240].Q THEN
       "Unit1.Em3.ControlNodes".topTapeLoading.sequence.status.nextStep := #JOB_2_STEP_50;
   END_IF;
END_REGION

REGION Network 21: Step[250] : Top Tape Cutter Clamp Down
   RUNG wire#powerrail
      { S7_Templates := "SrcType := DInt" } EQ_Contact(in1 := "Unit1.Em3.ControlNodes".topTapeLoading.sequence.status.currentStep, in2 := #JOB_2_STEP_50)
      Contact( "Unit1.Em3.ControlNodes".topTapeLoading.sequence.status.seqActive )
      wire#w1
      I_Contact( "Unit1.Em3.ControlNodes".cmTopTapeCutterClampUpDown.monitoring.inWorkPos )
      Coil( "Unit1.Em3.ControlNodes".topTapeLoading."step".action1[250] )
   END_RUNG
   RUNG wire#w1
      Contact( "Unit1.Em3.ControlNodes".cmTopTapeCutterClampUpDown.monitoring.inWorkPos )
      Coil( "Unit1.Em3.ControlNodes".topTapeLoading."step".transition1[250] )
   END_RUNG
   RUNG wire#w1
      Contact( "Unit1.Em3.ControlNodes".topTapeLoading."step".transition1[250] )
      { S7_Templates := "time_type := Time" } #statTonTime[250].TON(pt := T#500ms, et =>)
      Move(in := #JOB_2_STEP_60, out1 => "Unit1.Em3.ControlNodes".topTapeLoading.sequence.status.nextStep)
   END_RUNG
   // the same network as SCL:
   #_w1 := ("Unit1.Em3.ControlNodes".topTapeLoading.sequence.status.currentStep = #JOB_2_STEP_50) AND "Unit1.Em3.ControlNodes".topTapeLoading.sequence.status.seqActive;
   "Unit1.Em3.ControlNodes".topTapeLoading."step".action1[250] := #_w1 AND NOT "Unit1.Em3.ControlNodes".cmTopTapeCutterClampUpDown.monitoring.inWorkPos;
   "Unit1.Em3.ControlNodes".topTapeLoading."step".transition1[250] := #_w1 AND "Unit1.Em3.ControlNodes".cmTopTapeCutterClampUpDown.monitoring.inWorkPos;
   #statTonTime[250].TON(IN := #_w1 AND "Unit1.Em3.ControlNodes".topTapeLoading."step".transition1[250],
                         PT := T#500ms);
   IF #statTonTime[250].Q THEN
       "Unit1.Em3.ControlNodes".topTapeLoading.sequence.status.nextStep := #JOB_2_STEP_60;
   END_IF;
END_REGION

REGION Network 22: Step[260] : Top Tape Tension Backward
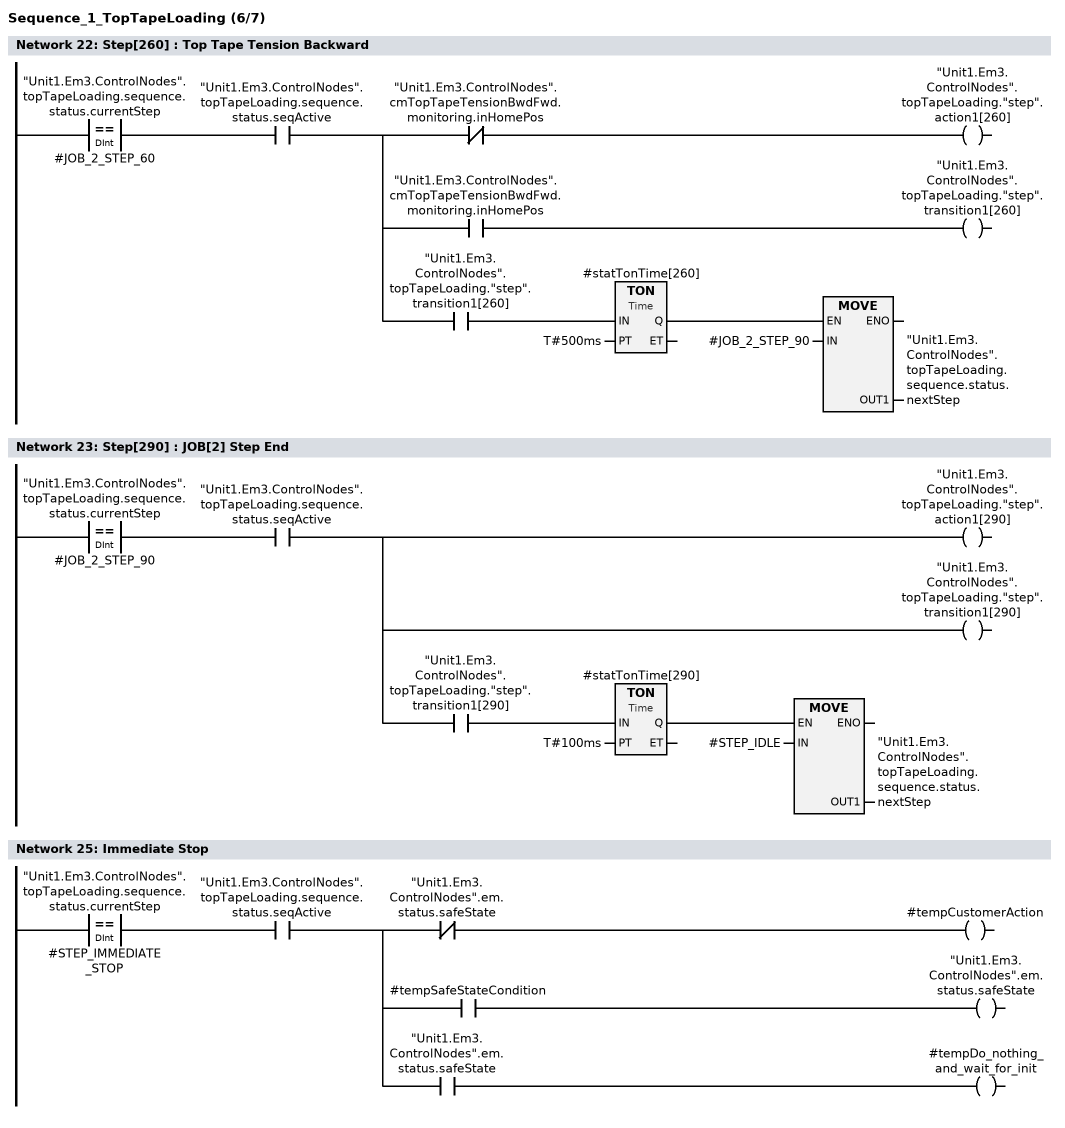
   RUNG wire#powerrail
      { S7_Templates := "SrcType := DInt" } EQ_Contact(in1 := "Unit1.Em3.ControlNodes".topTapeLoading.sequence.status.currentStep, in2 := #JOB_2_STEP_60)
      Contact( "Unit1.Em3.ControlNodes".topTapeLoading.sequence.status.seqActive )
      wire#w1
      I_Contact( "Unit1.Em3.ControlNodes".cmTopTapeTensionBwdFwd.monitoring.inHomePos )
      Coil( "Unit1.Em3.ControlNodes".topTapeLoading."step".action1[260] )
   END_RUNG
   RUNG wire#w1
      Contact( "Unit1.Em3.ControlNodes".cmTopTapeTensionBwdFwd.monitoring.inHomePos )
      Coil( "Unit1.Em3.ControlNodes".topTapeLoading."step".transition1[260] )
   END_RUNG
   RUNG wire#w1
      Contact( "Unit1.Em3.ControlNodes".topTapeLoading."step".transition1[260] )
      { S7_Templates := "time_type := Time" } #statTonTime[260].TON(pt := T#500ms, et =>)
      Move(in := #JOB_2_STEP_90, out1 => "Unit1.Em3.ControlNodes".topTapeLoading.sequence.status.nextStep)
   END_RUNG
   // the same network as SCL:
   #_w1 := ("Unit1.Em3.ControlNodes".topTapeLoading.sequence.status.currentStep = #JOB_2_STEP_60) AND "Unit1.Em3.ControlNodes".topTapeLoading.sequence.status.seqActive;
   "Unit1.Em3.ControlNodes".topTapeLoading."step".action1[260] := #_w1 AND NOT "Unit1.Em3.ControlNodes".cmTopTapeTensionBwdFwd.monitoring.inHomePos;
   "Unit1.Em3.ControlNodes".topTapeLoading."step".transition1[260] := #_w1 AND "Unit1.Em3.ControlNodes".cmTopTapeTensionBwdFwd.monitoring.inHomePos;
   #statTonTime[260].TON(IN := #_w1 AND "Unit1.Em3.ControlNodes".topTapeLoading."step".transition1[260],
                         PT := T#500ms);
   IF #statTonTime[260].Q THEN
       "Unit1.Em3.ControlNodes".topTapeLoading.sequence.status.nextStep := #JOB_2_STEP_90;
   END_IF;
END_REGION

REGION Network 23: Step[290] : JOB[2] Step End
   RUNG wire#powerrail
      { S7_Templates := "SrcType := DInt" } EQ_Contact(in1 := "Unit1.Em3.ControlNodes".topTapeLoading.sequence.status.currentStep, in2 := #JOB_2_STEP_90)
      Contact( "Unit1.Em3.ControlNodes".topTapeLoading.sequence.status.seqActive )
      wire#w1
      Coil( "Unit1.Em3.ControlNodes".topTapeLoading."step".action1[290] )
   END_RUNG
   RUNG wire#w1
      Coil( "Unit1.Em3.ControlNodes".topTapeLoading."step".transition1[290] )
   END_RUNG
   RUNG wire#w1
      Contact( "Unit1.Em3.ControlNodes".topTapeLoading."step".transition1[290] )
      { S7_Templates := "time_type := Time" } #statTonTime[290].TON(pt := T#100ms, et =>)
      Move(in := #STEP_IDLE, out1 => "Unit1.Em3.ControlNodes".topTapeLoading.sequence.status.nextStep)
   END_RUNG
   // the same network as SCL:
   "Unit1.Em3.ControlNodes".topTapeLoading."step".action1[290] := ("Unit1.Em3.ControlNodes".topTapeLoading.sequence.status.currentStep = #JOB_2_STEP_90) AND "Unit1.Em3.ControlNodes".topTapeLoading.sequence.status.seqActive;
   "Unit1.Em3.ControlNodes".topTapeLoading."step".transition1[290] := ("Unit1.Em3.ControlNodes".topTapeLoading.sequence.status.currentStep = #JOB_2_STEP_90) AND "Unit1.Em3.ControlNodes".topTapeLoading.sequence.status.seqActive;
   #statTonTime[290].TON(IN := ("Unit1.Em3.ControlNodes".topTapeLoading.sequence.status.currentStep = #JOB_2_STEP_90) AND "Unit1.Em3.ControlNodes".topTapeLoading.sequence.status.seqActive AND "Unit1.Em3.ControlNodes".topTapeLoading."step".transition1[290],
                         PT := T#100ms);
   IF #statTonTime[290].Q THEN
       "Unit1.Em3.ControlNodes".topTapeLoading.sequence.status.nextStep := #STEP_IDLE;
   END_IF;
END_REGION

REGION Network 24: *************** IMMEDIATE STOP ****************
END_REGION

REGION Network 25: Immediate Stop
   RUNG wire#powerrail
      { S7_Templates := "SrcType := DInt" } EQ_Contact(in1 := "Unit1.Em3.ControlNodes".topTapeLoading.sequence.status.currentStep, in2 := #STEP_IMMEDIATE_STOP)
      Contact( "Unit1.Em3.ControlNodes".topTapeLoading.sequence.status.seqActive )
      wire#w1
      I_Contact( "Unit1.Em3.ControlNodes".em.status.safeState )
      Coil( #tempCustomerAction )
   END_RUNG
   RUNG wire#w1
      Contact( #tempSafeStateCondition )
      Coil( "Unit1.Em3.ControlNodes".em.status.safeState )
   END_RUNG
   RUNG wire#w1
      Contact( "Unit1.Em3.ControlNodes".em.status.safeState )
      Coil( #tempDo_nothing_and_wait_for_init )
   END_RUNG
   // the same network as SCL:
   #_w1 := ("Unit1.Em3.ControlNodes".topTapeLoading.sequence.status.currentStep = #STEP_IMMEDIATE_STOP) AND "Unit1.Em3.ControlNodes".topTapeLoading.sequence.status.seqActive;
   #tempCustomerAction := #_w1 AND NOT "Unit1.Em3.ControlNodes".em.status.safeState;
   "Unit1.Em3.ControlNodes".em.status.safeState := #_w1 AND #tempSafeStateCondition;
   #tempDo_nothing_and_wait_for_init := #_w1 AND "Unit1.Em3.ControlNodes".em.status.safeState;
END_REGION

REGION Network 26: *************** STATUS **********************
END_REGION

REGION Network 27: Sequence Status
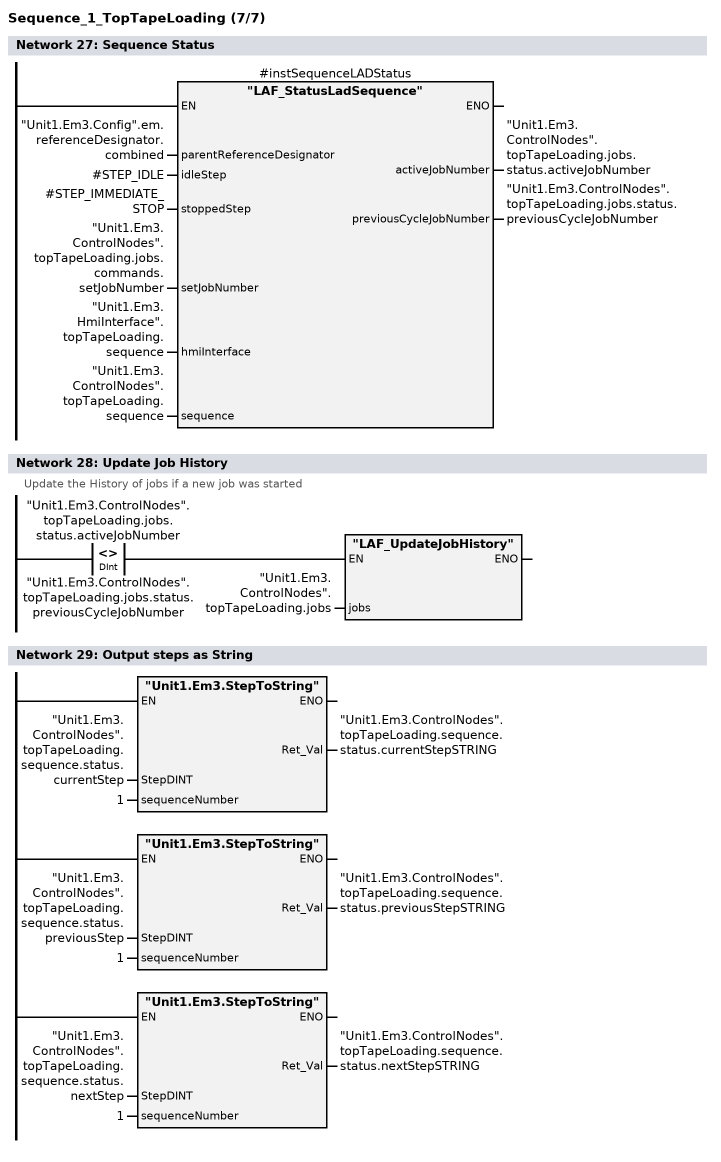
   RUNG wire#powerrail
      #instSequenceLADStatus(parentReferenceDesignator := "Unit1.Em3.Config".em.referenceDesignator.combined, idleStep := #STEP_IDLE, stoppedStep := #STEP_IMMEDIATE_STOP, setJobNumber := "Unit1.Em3.ControlNodes".topTapeLoading.jobs.commands.setJobNumber, hmiInterface := "Unit1.Em3.HmiInterface".topTapeLoading.sequence, sequence := "Unit1.Em3.ControlNodes".topTapeLoading.sequence, activeJobNumber => "Unit1.Em3.ControlNodes".topTapeLoading.jobs.status.activeJobNumber, previousCycleJobNumber => "Unit1.Em3.ControlNodes".topTapeLoading.jobs.status.previousCycleJobNumber)
   END_RUNG
   // the same network as SCL:
   #instSequenceLADStatus(parentReferenceDesignator := "Unit1.Em3.Config".em.referenceDesignator.combined,   // "LAF_StatusLadSequence"
                          idleStep := #STEP_IDLE,
                          stoppedStep := #STEP_IMMEDIATE_STOP,
                          setJobNumber := "Unit1.Em3.ControlNodes".topTapeLoading.jobs.commands.setJobNumber,
                          hmiInterface := "Unit1.Em3.HmiInterface".topTapeLoading.sequence,
                          sequence := "Unit1.Em3.ControlNodes".topTapeLoading.sequence,
                          activeJobNumber => "Unit1.Em3.ControlNodes".topTapeLoading.jobs.status.activeJobNumber,
                          previousCycleJobNumber => "Unit1.Em3.ControlNodes".topTapeLoading.jobs.status.previousCycleJobNumber);
END_REGION

REGION Network 28: Update Job History
   // Update the History of jobs if a new job was started
   RUNG wire#powerrail
      { S7_Templates := "SrcType := DInt" } NE_Contact(in1 := "Unit1.Em3.ControlNodes".topTapeLoading.jobs.status.activeJobNumber, in2 := "Unit1.Em3.ControlNodes".topTapeLoading.jobs.status.previousCycleJobNumber)
      "LAF_UpdateJobHistory"(jobs := "Unit1.Em3.ControlNodes".topTapeLoading.jobs)
   END_RUNG
   // the same network as SCL:
   IF "Unit1.Em3.ControlNodes".topTapeLoading.jobs.status.activeJobNumber <> "Unit1.Em3.ControlNodes".topTapeLoading.jobs.status.previousCycleJobNumber THEN
       "LAF_UpdateJobHistory"(jobs := "Unit1.Em3.ControlNodes".topTapeLoading.jobs);
   END_IF;
END_REGION

REGION Network 29: Output steps as String
   RUNG wire#powerrail
      "Unit1.Em3.StepToString"(StepDINT := "Unit1.Em3.ControlNodes".topTapeLoading.sequence.status.currentStep, sequenceNumber := 1, Ret_Val => "Unit1.Em3.ControlNodes".topTapeLoading.sequence.status.currentStepSTRING)
   END_RUNG
   RUNG wire#powerrail
      "Unit1.Em3.StepToString"(StepDINT := "Unit1.Em3.ControlNodes".topTapeLoading.sequence.status.previousStep, sequenceNumber := 1, Ret_Val => "Unit1.Em3.ControlNodes".topTapeLoading.sequence.status.previousStepSTRING)
   END_RUNG
   RUNG wire#powerrail
      "Unit1.Em3.StepToString"(StepDINT := "Unit1.Em3.ControlNodes".topTapeLoading.sequence.status.nextStep, sequenceNumber := 1, Ret_Val => "Unit1.Em3.ControlNodes".topTapeLoading.sequence.status.nextStepSTRING)
   END_RUNG
   // the same network as SCL:
   "Unit1.Em3.ControlNodes".topTapeLoading.sequence.status.currentStepSTRING := "Unit1.Em3.StepToString"(StepDINT := "Unit1.Em3.ControlNodes".topTapeLoading.sequence.status.currentStep,
                           sequenceNumber := 1);
   "Unit1.Em3.ControlNodes".topTapeLoading.sequence.status.previousStepSTRING := "Unit1.Em3.StepToString"(StepDINT := "Unit1.Em3.ControlNodes".topTapeLoading.sequence.status.previousStep,
                           sequenceNumber := 1);
   "Unit1.Em3.ControlNodes".topTapeLoading.sequence.status.nextStepSTRING := "Unit1.Em3.StepToString"(StepDINT := "Unit1.Em3.ControlNodes".topTapeLoading.sequence.status.nextStep,
                           sequenceNumber := 1);
END_REGION
END_FUNCTION_BLOCK
